TYPE ScaleFactor :
STRUCT
	MinFactor	: USINT; // Sensor Minimum Range
	MaxFactor	: USINT; // Sensor Maximum Range
END_STRUCT
END_TYPE

(* stored: Version 1.1.0.1, ProductVersion 3.1.4024.12
   DUT ScaleFactor: Id {1cd926df-6b68-4243-a994-ebb3f58e261d} *)
